SUBAPPLICATION Licht (* Subapplication Type *)
  (* Standard: 61499-2 *)
  (* Version 1.0, 2023-01-29, Franz *)
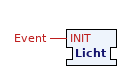
  EVENT_INPUT
    INIT; (* Service Initialization *)
  END_EVENT
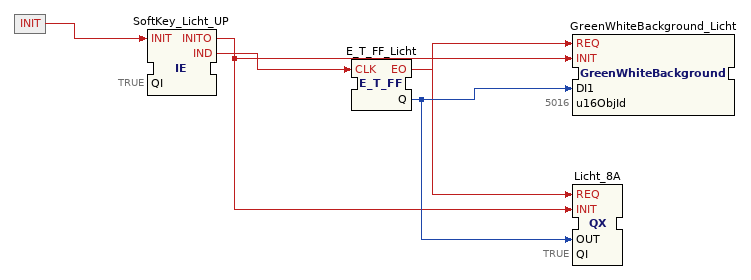
  FBS
    E_T_FF_Licht : E_T_FF;
    GreenWhiteBackground_Licht : GreenWhiteBackground(u16ObjId := 5016);
    Licht_8A : QX(QI := TRUE);
    SoftKey_Licht_UP : IE(QI := TRUE);
  END_FBS
  EVENT_CONNECTIONS
    E_T_FF_Licht.EO TO Licht_8A.REQ;
    E_T_FF_Licht.EO TO GreenWhiteBackground_Licht.REQ;
    INIT TO SoftKey_Licht_UP.INIT;
    SoftKey_Licht_UP.INITO TO GreenWhiteBackground_Licht.INIT;
    SoftKey_Licht_UP.INITO TO Licht_8A.INIT;
    SoftKey_Licht_UP.IND TO E_T_FF_Licht.CLK;
  END_CONNECTIONS
  DATA_CONNECTIONS
    E_T_FF_Licht.Q TO Licht_8A.OUT;
    E_T_FF_Licht.Q TO GreenWhiteBackground_Licht.DI1;
  END_CONNECTIONS
END_SUBAPPLICATION
